TYPE OutputBase_10CEE7DE :
STRUCT
END_STRUCT
END_TYPE

(* stored: Version 1.2.0.0, ProductVersion 3.1.4024.11
   DUT OutputBase_10CEE7DE: Id {06edf48d-f56b-45a6-aa78-7961b1df6b8f} *)
